FUNCTION_BLOCK PUBLIC PistonInsertStation
VAR_INPUT
END_VAR
VAR_OUTPUT
END_VAR
VAR
	xTrigger :BOOL := FALSE; // triggers processing
	State : ePistonInsertStaState := ePistonInsertStaState.eUnknown;
	NextState : ePistonInsertStaState := ePistonInsertStaState.eUnknown;
	ErrorReturnState : ePistonInsertStaState := ePistonInsertStaState.eUnknown;
	bFirst : BOOL := TRUE;
	VUT : BYTE; //VehicleID Under Station
	DwellTimer : TON;
	StateTimer : TON;
	PartPresentTimer : TON;
END_VAR

//////////////////// ESTOP TO STATION DISABLED
// If Piston Station is disabled, then we want to make sure that we have the SMC homed and not in the way of barrels
// we also want to check if the pallet hold downs and barrel backup position are correct
// if all above conditions are true, then we want to wait in a station disabled ready state
////////////////// STATION DISABLED - STATION ENABLED
// We have to go to have a piston ready for insertion, but also have operator hit start button
/////////////////////// STATION ENABLED - STATION DISABLED
// We have to go into disabled state
//////////////////////// ESTOP- STATION ENABLED
//// Follow all the logic to get the station ready

IF (GVL_IO.MachineEStopped) THEN 
	State := ePistonInsertStaState.eUnknown;
	NextState := ePistonInsertStaState.eUnknown;
	ErrorReturnState := ePistonInsertStaState.eUnknown;
	Status.PistonStatusMsg:= 'PistonSta Unknown, Check AIR, E-STOP and Hit Start';
END_IF

CASE State OF
	
ePistonInsertStaState.eUnknown:
    Status.PistonStatusMsg:= 'PistonSta Unknown, Check AIR, E-STOP and Hit Start';
	
    GVL_IO.PI_YMtrReset := FALSE; // we need a rising edge when we do a reset
	GVL_IO.PI_YMtrSetEnable:= FALSE; // we need a rising edge when we move to the Motor Reset State in the following states
	Act_SendEscapementtoWork();
	IF (GVL_IO.MC_XStartPB AND GVL_IO.MC_XAirPressureOK  AND GVL_IO.MC_NotEStopped) THEN // wait for start button when powered up or PLC program restarted ( remove this "TRUE" after debug
		ResetDwellTimer();
		ResetStateTimer();
		LEY_MasterReset();
        NextState := ePistonInsertStaState.eSMCMtrReset;		
	END_IF	

ePistonInsertStaState.eSMCMtrReset:
    DwellTimer(IN:= TRUE, PT:= T#1S);
	IF (DwellTimer.Q) THEN
		DwellTimer(IN:=FALSE);
		GVL_IO.PI_YMtrReset := NOT GVL_IO.PI_YMtrReset; // toggle the Reset to clear Alarms
	END_IF

	IF(NOT GVL_IO.PI_XMtrAlarm) THEN
		GVL_IO.PI_YMtrReset := FALSE;
        GVL_IO.PI_YMtrSetEnable := TRUE;
		ResetDwellTimer();
		NextState := ePistonInsertStaState.eSMCMtrCheckEnabled; // change to check enabled
	END_IF
	
	StateTimer(IN:= TRUE, PT:= T#10S);
	IF (StateTimer.Q) THEN
		ErrorReturnState := ePistonInsertStaState.eSMCMtrReset;
		Status.PistonStatusMsg:= 'Unable to Reset Piston Motor, Restart LEY controller';
		ResetDwellTimer();
		ResetStateTimer();
        NextState := ePistonInsertStaState.eError;		
	END_IF
	
	

ePistonInsertStaState.eSMCMtrCheckEnabled:
   IF (GVL_IO.PI_XMtrServoEnabled AND NOT GVL_IO.PI_XMtrBusy AND NOT GVL_IO.PI_XMtrEStopped AND NOT GVL_IO.PI_XMtrAlarm) THEN
	   NextState := ePistonInsertStaState.eSMCMtrSendHome;
	   ResetDwellTimer();
   END_IF
   DwellTimer(IN:=TRUE, PT:= T#10S);
   IF (DwellTimer.Q) THEN
		ErrorReturnState := ePistonInsertStaState.eUnknown;
		Status.PistonStatusMsg:= 'Unable to Enable Piston Motor, Restart LEY controller';
		ResetDwellTimer();
		ResetStateTimer();
        NextState := ePistonInsertStaState.eError;		
	END_IF
   
 ePistonInsertStaState.eSMCMtrSendHome:
	GVL_IO.PI_YMtrGoHome := TRUE;
	IF (GVL_IO.PI_XMtrServoHomed) THEN 
		NextState := ePistonInsertStaState.eSMCMtrHomed;
		GVL_IO.PI_YMtrGoHome := FALSE;
		ResetDwellTimer();
	END_IF
	DwellTimer(IN:=TRUE, PT:= T#10S);
	IF (DwellTimer.Q) THEN
		ErrorReturnState := ePistonInsertStaState.eUnknown;
		Status.PistonStatusMsg:= 'Unable to Home Piston Motor, Clear any jams ';
		ResetDwellTimer();
		ResetStateTimer();
        NextState := ePistonInsertStaState.eError;		
	END_IF   

	   
ePistonInsertStaState.eSMCMtrHomed:
     IF (GVL_IO.PI_XMtrServoHomed AND GVL_IO.PI_XMtrServoEnabled AND NOT GVL_IO.PI_XMtrBusy (*AND GVL_IO.PI_XMtrMoveCompl*) AND GVL_IO.PI_XMtrReady) THEN
		 NextState := ePistonInsertStaState.eInit;  // not checking tool position in IMBAD2
		 ResetDwellTimer();	 
	 END_IF
	 
	DwellTimer(IN:=TRUE, PT:= T#10S);
	IF (DwellTimer.Q) THEN
		ErrorReturnState := ePistonInsertStaState.eUnknown;
		Status.PistonStatusMsg:= 'Unable to Ready Piston Motor, Restart LEY ';
		ResetDwellTimer();
		ResetStateTimer();
        NextState := ePistonInsertStaState.eError;		
	END_IF   


ePistonInsertStaState.eCheckToolPosition:
	IF (LotsData.Lot.BarrelSize = eBarrelType.Size55cc) THEN
		IF (TRUE OR GVL_IO.PI_XToolAt55_10_Barrel AND NOT GVL_IO.PI_XToolAt3_30_Barrel) THEN // no barrel backup 
			 NextState := ePistonInsertStaState.eInit;
		ELSE
			NextState := ePistonInsertStaState.eUnknown;
       		Status.PistonStatusMsg:= 'Incorrect Backup Location,Fix and Hit Start';
		END_IF
	ELSIF (LotsData.Lot.BarrelSize = eBarrelType.Size30cc) THEN
		IF (TRUE OR NOT GVL_IO.PI_XToolAt55_10_Barrel AND GVL_IO.PI_XToolAt3_30_Barrel) THEN
			 NextState := ePistonInsertStaState.eInit;
		ELSE
			NextState := ePistonInsertStaState.eUnknown;
        	Status.PistonStatusMsg:= 'Incorrect Backup Location,Fix and Hit Start';
		END_IF
	ELSE 
		NextState := ePistonInsertStaState.eUnknown;
        Status.PistonStatusMsg:= 'Incorrect Part Selection, Start New Lot';
	END_IF
	

ePistonInsertStaState.eInit:
	Act_RetractBarrelBackup();    
	Act_FreePalletHoldDown();	
	IF (GVL_IO.PI_XPistonPresentEscapement) THEN
		Act_SendEscapementtoWork();        
    ELSE 
		Act_SendEscapementToBowl();
	END_IF		
	ResetDwellTimer();
	NextState := ePistonInsertStaState.eHoming;

ePistonInsertStaState.eHoming:
    IF(IsBarrelBackupRetracted() AND IsPalletHoldDownFree()) THEN   
		ResetDwellTimer();
	 	IF (GVL_IO.PI_YEscapementToBowl) THEN // based on what direction decided in previous state
			NextState := ePistonInsertStaState.eMoveEscapemttoBowl;	
		ELSE
			NextState := ePistonInsertStaState.eMoveEscapmentToWork;
		END_IF		
	    IF (NOT LotsData.Lot.PistonInsertEnabled) THEN
			NextState := ePistonInsertStaState.eDisabledReady;
        END_IF	
	END_IF
	
	DwellTimer(IN:=TRUE, PT:= T#10S);
	IF (DwellTimer.Q) THEN
		ErrorReturnState := ePistonInsertStaState.eInit;		
		ResetDwellTimer();
		ResetStateTimer();
        NextState := ePistonInsertStaState.eError;		
	END_IF   

	
ePistonInsertStaState.eDisabledReady:
  IF (LotsData.Lot.PistonInsertEnabled) THEN
	  NextState := ePistonInsertStaState.eUnknown;
  END_IF
  IF (xTrigger) THEN
	  NextState := ePistonInsertStaState.eDepart;
  END_IF
  Status.PistonStatusMsg:= 'Station Disabled and Ready';


ePistonInsertStaState.eMoveEscapemttoBowl:
  	Act_SendEscapementToBowl();    
  	IF (IsEscapementAtBowl()) THEN
		ResetDwellTimer();
	  	NextState := ePistonInsertStaState.eEscapmentAtBowl;
  	END_IF
	
	DwellTimer(IN:=TRUE, PT:= T#10S);
	IF (DwellTimer.Q) THEN
		ErrorReturnState := ePistonInsertStaState.eMoveEscapemttoBowl;
		Status.PistonStatusMsg:= 'Escapement unable to move to Bowl,Stuck Pistons?';
		ResetDwellTimer();
		ResetStateTimer();
        NextState := ePistonInsertStaState.eError;		
	END_IF   
 
	
	 
ePistonInsertStaState.eEscapmentAtBowl:
	NextState := ePistonInsertStaState.eWaitForPartAtBowl;
	PartPresentTimer(IN:=FALSE);
	DwellTimer(IN:=FALSE);
	StateTimer(IN:=FALSE);

ePistonInsertStaState.eWaitForPartAtBowl:
    PartPresentTimer(IN:= GVL_IO.PI_XPistonPresentEscapement, PT := T#10MS); //uncommented FOR turnkey debug
	//PartPresentTimer(IN:= TRUE, PT := T#10MS); //comment this out later
    IF (PartPresentTimer.Q) THEN
		PartPresentTimer(IN:=FALSE);
		NextState := ePistonInsertStaState.eMoveEscapmentToWork;
		StateTimer(IN:=FALSE);
        ResetDwellTimer();		
	END_IF	
	
    DwellTimer(IN:=TRUE, PT:= T#10S);
	IF (DwellTimer.Q) THEN
		ErrorReturnState := ePistonInsertStaState.eMoveEscapemttoBowl;
		Status.PistonStatusMsg:= 'Piston: No Piston Detected. Is Bowl Empty? ';
		ResetDwellTimer();
		ResetStateTimer();
        NextState := ePistonInsertStaState.eError;		
	END_IF   

ePistonInsertStaState.eMoveEscapmentToWork:
 	Act_SendEscapementtoWork();
	IF (IsEscapementAtWork()) THEN
		ResetDwellTimer();
		NextState := ePistonInsertStaState.eEscapementAtWork;
	END_IF
	
	DwellTimer(IN:=TRUE, PT:= T#10S);
	IF (DwellTimer.Q) THEN
		ErrorReturnState := ePistonInsertStaState.eMoveEscapmentToWork;
		Status.PistonStatusMsg:= 'Escapement Slide Failed to go to Work';
		ResetDwellTimer();
		ResetStateTimer();
        NextState := ePistonInsertStaState.eError;		
	END_IF   


ePistonInsertStaState.eEscapementAtWork:	
	NextState := ePistonInsertStaState.eReady; // We have captured a part and now sitting on top of the motor shaft waiting for the vehicle to arrive
	

ePistonInsertStaState.eReady: // vehicle arrives to station 
	IF (xTrigger) THEN
		Act_EngagePalletHoldDown();
		Act_ExtendBarrelBackup();
		ResetDwellTimer();
        NextState := ePistonInsertStaState.ePalletHoldDownEngaged;		
		PartsData.Status[VUT].OverallStatus := ePartStatus.eReject; //define as reject upfront, later update status	          		
	END_IF
	Status.PistonStatusMsg:= 'Waiting For Vehicle To Process';

ePistonInsertStaState.ePalletHoldDownEngaged:
   Act_EngagePalletHoldDown();
   IF (IsPalletHoldDownEngaged()) THEN
	   Act_ExtendBarrelBackup();
	   ResetDwellTimer();
       NextState := ePistonInsertStaState.eWaitForBarrelBackupEngaged;   
   END_IF
   
   DwellTimer(IN:=TRUE, PT:= T#10S);
	IF (DwellTimer.Q) THEN
		ErrorReturnState := ePistonInsertStaState.ePalletHoldDownEngaged;		
		ResetDwellTimer();
		ResetStateTimer();
        NextState := ePistonInsertStaState.eError;		
	END_IF   
   
   
ePistonInsertStaState.eWaitForBarrelBackupEngaged:
	IF(IsBarrelBackupExtended()) THEN
		ResetDwellTimer();
		NextState := ePistonInsertStaState.eFirePistonUp;
	END_IF
  
	DwellTimer(IN:=TRUE, PT:= T#10S);
	IF (DwellTimer.Q) THEN
		ErrorReturnState := ePistonInsertStaState.ePalletHoldDownEngaged;		
		ResetDwellTimer();
		ResetStateTimer();
        NextState := ePistonInsertStaState.eError;		
	END_IF   

ePistonInsertStaState.eFirePistonUp:
    IF (LotsData.Lot.BarrelSize = eBarrelType.Size10cc) THEN // program 1 = 10cc
    	GVL_IO.PI_YMtrStepSelectIN0 := TRUE;
		GVL_IO.PI_YMtrStepSelectIN1 := FALSE;
	ELSIF (LotsData.Lot.BarrelSize = eBarrelType.Size5cc) THEN //program3 = 5 cc
		GVL_IO.PI_YMtrStepSelectIN0 := TRUE;
		GVL_IO.PI_YMtrStepSelectIN1 := TRUE;
	ELSE // must be 3 cc 
		GVL_IO.PI_YMtrStepSelectIN0 := FALSE; //program2 = 3cc
		GVL_IO.PI_YMtrStepSelectIN1 := TRUE;
	END_IF
	DwellTimer(IN:=TRUE,PT:= T#20MS);
	IF(DwellTimer.Q) THEN
		DwellTimer(IN:=FALSE);
		GVL_IO.PI_YMtrDriveStepTrigger:= TRUE;
		NextState := ePistonInsertStaState.eWaitForPistonStartMovUp;
	END_IF

ePistonInsertStaState.eWaitForPistonStartMovUp:
	 IF (NOT GVL_IO.PI_XMtrMoveCompl) THEN   //Piston has started to move up
		 GVL_IO.PI_YMtrDriveStepTrigger:= FALSE;
		 GVL_IO.PI_YMtrStepSelectIN0 := FALSE;
		 GVL_IO.PI_YMtrStepSelectIN1 := FALSE;
		 ResetDwellTimer();
		 NextState := ePistonInsertStaState.eWaitForPistonMovDoneUp;
	 END_IF
	DwellTimer(IN:=TRUE, PT:= T#10S);
	IF (DwellTimer.Q) THEN
		ErrorReturnState := ePistonInsertStaState.eFirePistonUp;		
		GVL_IO.PI_YMtrDriveStepTrigger:= FALSE;
		ResetDwellTimer();
		ResetStateTimer();
		Status.PistonStatusMsg:= 'SMC Mtr Possibly Jammed, Lock I/O and Home Mtr';
        NextState := ePistonInsertStaState.eError;		
	END_IF 


ePistonInsertStaState.eWaitForPistonMovDoneUp:
 	IF (GVL_IO.PI_XMtrMoveCompl) THEN
		NextState := ePistonInsertStaState.eFirePistonDown;    //There may be a way to read piston actual position
		ResetDwellTimer();
		UpdatePartData();
 	END_IF
 	DwellTimer(IN:=TRUE, PT:= T#10S);
	IF (DwellTimer.Q) THEN
		ErrorReturnState := ePistonInsertStaState.eFirePistonUp;		
		GVL_IO.PI_YMtrDriveStepTrigger:= FALSE;
		ResetDwellTimer();
		ResetStateTimer();
		Status.PistonStatusMsg:= 'SMC Mtr Possibly Jammed, Lock I/O and Home Mtr';
        NextState := ePistonInsertStaState.eError;		
	END_IF 
 

ePistonInsertStaState.eFirePistonDown:
	GVL_IO.PI_YMtrStepSelectIN0 := FALSE;
	GVL_IO.PI_YMtrStepSelectIN1 := FALSE;
	GVL_IO.PI_YMtrDriveStepTrigger:= TRUE;
	ResetDwellTimer();
	NextState := ePistonInsertStaState.eWaitForPistonStartMovDwn;

ePistonInsertStaState.eWaitForPistonStartMovDwn:
 	IF (NOT GVL_IO.PI_XMtrMoveCompl) THEN
		GVL_IO.PI_YMtrDriveStepTrigger:= FALSE;
		GVL_IO.PI_YMtrStepSelectIN0 := FALSE;
		GVL_IO.PI_YMtrStepSelectIN1 := FALSE;
		ResetDwellTimer();
	 	NextState := ePistonInsertStaState.eWaitForPistonMovDoneDown;
 	END_IF
	
	DwellTimer(IN:=TRUE, PT:= T#10S);
	IF (DwellTimer.Q) THEN
		ErrorReturnState := ePistonInsertStaState.eFirePistonDown;		
		GVL_IO.PI_YMtrDriveStepTrigger:= FALSE;
		ResetDwellTimer();
		ResetStateTimer();
		Status.PistonStatusMsg:= 'SMC Mtr Possibly Jammed, Lock I/O and Home Mtr';
        NextState := ePistonInsertStaState.eError;		
	END_IF 
  


ePistonInsertStaState.eWaitForPistonMovDoneDown:	
 	IF (GVL_IO.PI_XMtrMoveCompl) THEN
		NextState := ePistonInsertStaState.eRetractPalletHoldDownAndBarrel;
		ResetDwellTimer();
 	END_IF
	//Act_FreePalletHoldDown();   // removed at Turnkey because piston gets jammed
	//Act_RetractBarrelBackup();
	
    DwellTimer(IN:=TRUE, PT:= T#10S);
	IF (DwellTimer.Q) THEN
		ErrorReturnState := ePistonInsertStaState.eFirePistonDown;		
		GVL_IO.PI_YMtrDriveStepTrigger:= FALSE;
		ResetDwellTimer();
		ResetStateTimer();
		Status.PistonStatusMsg:= 'SMC Mtr Possibly Jammed, Lock I/O and Home Mtr';
        NextState := ePistonInsertStaState.eError;		
	END_IF 
	

 
 ePistonInsertStaState.eRetractPalletHoldDownAndBarrel:
 	Act_FreePalletHoldDown();
	Act_RetractBarrelBackup();
	ResetDwellTimer();
	NextState := ePistonInsertStaState.eWaitForPalletHoldDownAndBackupRetracted; 
 
 ePistonInsertStaState.eWaitForPalletHoldDownAndBackupRetracted:
 	IF (IsBarrelBackUpRetracted() AND IsPalletHoldDownFree()) THEN
		ResetDwellTimer();
		ResetStateTimer();
		NextState := ePistonInsertStaState.eDepart;
 	END_IF
    
    DwellTimer(IN:=TRUE, PT:= T#10S);
	IF (DwellTimer.Q) THEN
		ErrorReturnState := ePistonInsertStaState.eRetractPalletHoldDownAndBarrel;		
		ResetDwellTimer();
		ResetStateTimer();
		NextState := ePistonInsertStaState.eError;		
	END_IF 
  

ePistonInsertStaState.eDepart:
	StateTimer(IN:=TRUE, PT:= T#20MS);
	IF (StateTimer.Q) THEN
		Stations.fbRoutePlanner.M_NotifyVehStaCmpl(StationIndex:= MM_CONST.PISTON_STA, VehicleID := VUT);
		xTrigger := FALSE;	
		StateTimer(IN:=FALSE);
		IF (NOT Stations.fbCycleControl.StopRequested) THEN			
			NextState := ePistonInsertStaState.eInit;
		ELSE 
			NextState := ePistonInsertStaState.eStopActive;
		END_IF
	END_IF

ePistonInsertStaState.eStopActive:
IF (NOT Stations.fbCycleControl.StopRequested) THEN			
	NextState := ePistonInsertStaState.eInit;
END_IF	
Status.PistonStatusMsg:= 'Piston Sta Cycle Stop, Hit Start'; 
	
ePistonInsertStaState.eError:
	Status.StationStauts[MM_CONST.PISTON_STA_HMI_STATE] := OverallStationStatus.eError;
	IF (GVL_IO.MC_XStartPB) THEN
		NextState := ErrorReturnState;
		ErrorReturnState := ePistonInsertStaState.eUnknown;
	END_IF

END_CASE

IF (State <> NextState) THEN
	bFirst := TRUE;
	StateTimer(IN:=FALSE);
ELSE
	bFirst := FALSE;
END_IF

State := NextState;
AssignStationStatusForHMI();

ACTION Act_EngagePalletHoldDown:
GVL_IO.PI_YPalletHoldDownExtend:= TRUE;
GVL_IO.PI_YPalletHoldDownRetract := FALSE;
END_ACTION

ACTION Act_ExtendBarrelBackup:
GVL_IO.PI_YBarrelBackupExtend := TRUE;
GVL_IO.PI_YBarrelBackupRetract := FALSE;
END_ACTION

ACTION Act_FreePalletHoldDown:
GVL_IO.PI_YPalletHoldDownExtend:= FALSE;
GVL_IO.PI_YPalletHoldDownRetract := TRUE;
END_ACTION

ACTION Act_RetractBarrelBackup:
GVL_IO.PI_YBarrelBackupExtend := FALSE;
GVL_IO.PI_YBarrelBackupRetract := TRUE;
END_ACTION

ACTION Act_SendEscapementToBowl:
GVL_IO.PI_YEscapementToBowl := TRUE;
GVL_IO.PI_YEscapementToWork := FALSE;
END_ACTION

ACTION Act_SendEscapementtoWork:
GVL_IO.PI_YEscapementToBowl := FALSE;
GVL_IO.PI_YEscapementToWork := TRUE;
END_ACTION

METHOD PUBLIC AssignStationStatusForHMI : BOOL
VAR_INPUT
END_VAR
Status.StationsState[MM_CONST.PISTON_STA_HMI_STATE] := State;
IF (NOT LotsData.Lot.PistonInsertEnabled AND NOT (State = ePistonInsertStaState.eUnknown) AND NOT (State = ePistonInsertStaState.eError)) THEN
	Status.StationStauts[MM_CONST.PISTON_STA_HMI_STATE] := OverallStationStatus.eDisabled;
ELSE 
	CASE State OF 
	ePistonInsertStaState.eUnknown,ePistonInsertStaState.eError: 
		Status.StationStauts[MM_CONST.PISTON_STA_HMI_STATE] := OverallStationStatus.eError;
	 
    
    ePistonInsertStaState.eSMCMtrReset,ePistonInsertStaState.eSMCMtrCheckEnabled,ePistonInsertStaState.eSMCMtrSendHome,
    ePistonInsertStaState.eSMCMtrHomed,ePistonInsertStaState.eInit, ePistonInsertStaState.eHoming,
	ePistonInsertStaState.eMoveEscapemttoBowl,
	ePistonInsertStaState.eEscapmentAtBowl,
	ePistonInsertStaState.eMoveEscapmentToWork,
	ePistonInsertStaState.eEscapementAtWork:
    	Status.StationStauts[MM_CONST.PISTON_STA_HMI_STATE] := OverallStationStatus.eHoming;	
	
	ePistonInsertStaState.eWaitForPartAtBowl:
		Status.StationStauts[MM_CONST.PISTON_STA_HMI_STATE] := OverallStationStatus.eWarning;
	
	ePistonInsertStaState.eReady:
		Status.StationStauts[MM_CONST.PISTON_STA_HMI_STATE] := OverallStationStatus.eWaitingForParts;
	
	ePistonInsertStaState.ePalletHoldDownEngaged,
	ePistonInsertStaState.eFirePistonUp,
	ePistonInsertStaState.eSendBarrelBackupEngage,
	ePistonInsertStaState.eWaitForPistonStartMovUp,
	ePistonInsertStaState.eWaitForBarrelBackupEngaged,
	ePistonInsertStaState.eWaitForPistonMovDoneUp,
	ePistonInsertStaState.eFirePistonDown,
	ePistonInsertStaState.eRetractPalletHoldDownAndBackup,
	ePistonInsertStaState.eWaitForPistonStartMovDwn,
	ePistonInsertStaState.eRetractPalletHoldDownAndBarrel,
	ePistonInsertStaState.eWaitForPalletHoldDownAndBackupRetracted,
	ePistonInsertStaState.eWaitForPistonMovDoneDown :
		Status.StationStauts[MM_CONST.PISTON_STA_HMI_STATE] := OverallStationStatus.eWaitingForParts; 
	
    ePistonInsertStaState.eStopActive:
	    Status.StationStauts[MM_CONST.PISTON_STA_HMI_STATE] := OverallStationStatus.eCycleStop;
	 
	ELSE ;
	
	END_CASE
END_IF
END_METHOD

METHOD PUBLIC ClearVehicleTrigger : BOOL
VAR_INPUT
END_VAR
xTrigger := FALSE;
END_METHOD

METHOD PUBLIC IsBarrelBackupExtended : BOOL
VAR_INPUT
END_VAR
IsBarrelBackUpExtended := TRUE;  // IMBAD 2 Has No Barrel Backup
(*
IsBarrelBackUpExtended := GVL_IO.PI_XBarrelHoldDownExtended AND NOT GVL_IO.PI_XBarrelHoldDownHome;
IF (NOT IsBarrelBackUpExtended) THEN
	Status.PistonStatusMsg := 'Piston: Check Barrel Backup Sensors';
END_IF
*)
END_METHOD

METHOD PUBLIC IsBarrelBackUpRetracted : BOOL
VAR_INPUT
END_VAR
IsBarrelBackUpRetracted := TRUE;  // IMBAD 2 has no Barrel Backup
(* 
IsBarrelBackUpRetracted := NOT GVL_IO.PI_XBarrelHoldDownExtended AND GVL_IO.PI_XBarrelHoldDownHome;
IF (NOT IsBarrelBackUpRetracted) THEN
	Status.PistonStatusMsg := 'Piston: Check Barrel Backup Sensors';
END_IF
*)
END_METHOD

METHOD PUBLIC IsEscapementAtBowl : BOOL
VAR_INPUT
END_VAR
IsEscapementAtBowl := (GVL_IO.PI_XEscapementAtBowl);// AND NOT GVL_IO.PI_XEscapementAtInsertLoc);
IF (NOT IsEscapementAtBowl) THEN
	Status.PistonStatusMsg := 'Piston: Check Escapment Sensors';
END_IF
END_METHOD

METHOD PUBLIC IsEscapementAtWork : BOOL
VAR_INPUT
END_VAR
IsEscapementAtWork := ((*NOT GVL_IO.PI_XEscapementAtBowl AND *)GVL_IO.PI_XEscapementAtInsertLoc);
IF (NOT IsEscapementAtWork) THEN
	Status.PistonStatusMsg := 'Piston: Check Escapment Sensors';
END_IF
END_METHOD

METHOD PUBLIC IsFaulted : BOOL
VAR_INPUT
END_VAR
IsFaulted := (State = ePistonInsertStaState.eUnknown OR State = ePistonInsertStaState.eError);
END_METHOD

METHOD PUBLIC IsPalletHoldDownEngaged : BOOL
VAR_INPUT
END_VAR
IsPalletHoldDownEngaged := (NOT GVL_IO.PI_XPalletHoldDownHome (*AND GVL_IO.PI_XPalletHoldDownExtended*));
IF (NOT IsPalletHoldDownEngaged) THEN
	Status.PistonStatusMsg := 'Piston: Check Pallet Hold Down'; 
END_IF
END_METHOD

METHOD PUBLIC IsPalletHoldDownFree : BOOL
VAR_INPUT
END_VAR
IsPalletHoldDownFree := (GVL_IO.PI_XPalletHoldDownHome AND NOT GVL_IO.PI_XPalletHoldDownExtended);
IF (NOT IsPalletHoldDownFree) THEN
	Status.PistonStatusMsg := 'Piston: Check Pallet Hold Down'; 
END_IF
END_METHOD

METHOD PUBLIC LEY_MasterReset : BOOL
VAR_INPUT
END_VAR
GVL_IO.PI_YMtrReset := TRUE;
GVL_IO.PI_YMtrSetEnable:= TRUE;
GVL_IO.PI_YMtrDriveStepTrigger := FALSE;
GVL_IO.PI_YMtrHoldMove := FALSE;
GVL_IO.PI_YMtrGoHome := FALSE;
GVL_IO.PI_YMtrJogNeg := FALSE;
GVL_IO.PI_YMtrJogPos := FALSE;
GVL_IO.PI_YMtrSwitchJogInch := FALSE;
GVL_IO.PI_YMtrStepSelectIN0:= FALSE;
GVL_IO.PI_YMtrStepSelectIN1:= FALSE;
GVL_IO.PI_YMtrStepSelectIN2:= FALSE;
GVL_IO.PI_YMtrStepSelectIN3:= FALSE;
GVL_IO.PI_YMtrStepSelectIN4:= FALSE;
GVL_IO.PI_YMtrStepSelectIN5:= FALSE;
END_METHOD

PROPERTY PUBLIC Ready : BOOL
GET
IF (LotsData.Lot.PistonInsertEnabled) THEN
	Ready := (State = ePistonInsertStaState.eReady);
ELSE
    Ready := (State = ePistonInsertStaState.eDisabledReady);
END_IF
END_GET
END_PROPERTY

ACTION ResetDwellTimer:
DwellTimer(IN:=FALSE);
END_ACTION

METHOD PUBLIC ResetState : BOOL
VAR_INPUT
END_VAR
	State := ePistonInsertStaState.eUnknown;
	NextState := ePistonInsertStaState.eUnknown;
END_METHOD

ACTION ResetStateTimer:
StateTimer(IN:=FALSE);
END_ACTION

PROPERTY PUBLIC Trigger : BOOL
SET
xTrigger := Trigger;
END_SET
END_PROPERTY

METHOD PUBLIC UpdatePartData : BOOL
VAR_INPUT
END_VAR
PartsData.Status[VUT].OverallStatus := ePartStatus.ePistonInserted;
PartsData.Status[VUT].PistonStroke := GVL_IO.PI_XMtrCurrPos;
PartsData.Status[VUT].PistonPass := TRUE;
PartsData.Status[VUT].PistonInsertTime := SYSTEMTIME_TO_STRING(Logging.fbCurrTime.systemTime);
END_METHOD

PROPERTY PUBLIC VehicleUnderTest : BYTE
GET
VehicleUnderTest := VUT;
END_GET
SET
VUT := VehicleUnderTest;
END_SET
END_PROPERTY

END_FUNCTION_BLOCK

(* stored: Version 1.1.0.1, ProductVersion 3.1.4022.6
   POU PistonInsertStation: Id {a02d9d91-336e-4478-b9fd-491c85696e9b}, SpecialFunc None
   Action Act_EngagePalletHoldDown: Id {56c1c9e5-497b-4f57-95ac-d0fe63cd6697}
   Action Act_ExtendBarrelBackup: Id {59448d0f-e721-42d6-9080-a9c6c45b6348}
   Action Act_FreePalletHoldDown: Id {4de681fd-280a-4937-b7fa-916e056184eb}
   Action Act_RetractBarrelBackup: Id {7dd7d522-98fe-486b-a58a-f11b0f0b76ed}
   Action Act_SendEscapementToBowl: Id {621cc3e8-4b67-4ffe-a537-877dce92507a}
   Action Act_SendEscapementtoWork: Id {e94132a5-3478-4bac-b294-f527b2a216e6}
   Method AssignStationStatusForHMI: Id {5a7326e4-aedc-44e6-b1d4-575423dcb9e7}
   Method ClearVehicleTrigger: Id {36dac945-390f-49e0-a2aa-0ec30dc03fc2}
   Method IsBarrelBackupExtended: Id {77d91311-7f03-4510-a220-fe912a5a1ad4}
   Method IsBarrelBackUpRetracted: Id {8db7cb75-5728-4a43-9927-279eb0e83ff3}
   Method IsEscapementAtBowl: Id {7c0fa6e7-01d9-41af-b14b-987e8a39ba3d}
   Method IsEscapementAtWork: Id {a9c38715-9e01-464f-819c-9ca739f09f45}
   Method IsFaulted: Id {f60b070c-dad7-45f0-ad11-b5b8e16bc359}
   Method IsPalletHoldDownEngaged: Id {30c9cd93-0b07-407c-853e-2e9026dbe0f7}
   Method IsPalletHoldDownFree: Id {09776c1e-b255-45db-b025-072113e799b8}
   Method LEY_MasterReset: Id {25262eea-0509-4e29-9e49-a0894fa697ac}
   Property Ready: Id {eafe2669-ae84-4b00-8e99-42736ebd354a}
   Get Get: Id {b1577c0a-e4ac-4d5d-9b28-6eaf8f39781e}
   Action ResetDwellTimer: Id {154bc63a-2b0d-4c6d-a076-47fb7f7725a8}
   Method ResetState: Id {36e9b148-74e7-48b7-83f7-a3e19f3ec41f}
   Action ResetStateTimer: Id {8e6b54b2-f47b-49a0-ba67-4d758d0f314b}
   Property Trigger: Id {52097ca3-d6f0-48ee-8cdf-03782f2030d0}
   Set Set: Id {0d134f10-d65f-44d9-9c3b-7f8c65fed1e4}
   Method UpdatePartData: Id {dc1dfcab-6b7c-4e28-986b-ce41d7c1cf6b}
   Property VehicleUnderTest: Id {97a15262-4287-4cb1-b64a-cd54823e6458}
   Get Get: Id {0ab11653-eb63-444f-81d2-17dc557f5264}
   Set Set: Id {9300343e-c948-4058-9a47-adccda4342a7} *)
